// TIA Portal V17 export
// export: Created 2025-06-20T11:32:37.9239786Z, ExportSetting WithDefaults, DisplayName Totally Integrated Automation Portal, DisplayVersion V17 Update 8, DisplayName TIA Portal Openness, DisplayVersion V17 Update 8, DisplayName TIA Portal Version Control Interface, DisplayVersion V17, DisplayName SINAMICS Startdrive Advanced, DisplayVersion V17 SP2, DisplayName SINAMICS Startdrive G110M, G120, G120C, G120D, G120P, G115D, DisplayVersion V17 SP2, DisplayName SINAMICS Startdrive G130, G150, S120, S150, SINAMICS MV, S210, DisplayVersion V17 SP2, DisplayName STEP 7 Professional, DisplayVersion V17 Update 8, DisplayName SINUMERIK ONE STEP 7 Toolbox, DisplayVersion V17 Update 12, DisplayName SINUMERIK ONE PLC Basic Program Plus, DisplayVersion V17 Update 12, DisplayName SINUMERIK 840D sl STEP 7 Toolbox, DisplayVersion V17 Update 12, DisplayName STEP 7 Safety, DisplayVersion V17 Update 6, DisplayName WinCC Advanced, DisplayVersion V17 Update 8
DATA_BLOCK "DB16500_CONNECTION_CALL_MON"   // DB16500
{ S7_Optimized_Access := 'FALSE'; DB_Accessible_From_OPC_UA := 'FALSE' }
VERSION : 0.1
// stored: AutoNumber false, DBAccessibleFromOPCUA false, DBAccessibleFromWebserver false, IsOnlyStoredInLoadMemory false, IsWriteProtectedInAS false
   VAR
      UNIT_1 : Struct
         STA_3_MEAS : Struct
            METHOD : Struct
               NOZZLE_SURFACE_DISTANCE : Struct
                  STATUS : DWord;
                  Connect : DWord;
                  NamespaceGetIndexList : DWord;
                  MethodGetHandleList : DWord;
                  MethodCall : DWord;
                  MethodReleaseHandleList : DWord;
                  Disconnect : DWord;
                  ConnectionGetStatus : DWord;
               END_STRUCT;
               START_LAYER_THICKNESS : Struct
                  STATUS : DWord;
                  Connect : DWord;
                  NamespaceGetIndexList : DWord;
                  MethodGetHandleList : DWord;
                  MethodCall : DWord;
                  MethodReleaseHandleList : DWord;
                  Disconnect : DWord;
                  ConnectionGetStatus : DWord;
               END_STRUCT;
               STOP_LAYER_THICKNESS : Struct
                  STATUS : DWord;
                  Connect : DWord;
                  NamespaceGetIndexList : DWord;
                  MethodGetHandleList : DWord;
                  MethodCall : DWord;
                  MethodReleaseHandleList : DWord;
                  Disconnect : DWord;
                  ConnectionGetStatus : DWord;
               END_STRUCT;
               CALIBRATING : Struct
                  STATUS : DWord;
                  Connect : DWord;
                  NamespaceGetIndexList : DWord;
                  MethodGetHandleList : DWord;
                  MethodCall : DWord;
                  MethodReleaseHandleList : DWord;
                  Disconnect : DWord;
                  ConnectionGetStatus : DWord;
               END_STRUCT;
               RESET : Struct
                  STATUS : DWord;
                  Connect : DWord;
                  NamespaceGetIndexList : DWord;
                  MethodGetHandleList : DWord;
                  MethodCall : DWord;
                  MethodReleaseHandleList : DWord;
                  Disconnect : DWord;
                  ConnectionGetStatus : DWord;
               END_STRUCT;
               READ_VARIABLES : Struct
                  STATUS : DWord;
                  Connect : DWord;
                  NamespaceGetIndexList : DWord;
                  MethodGetHandleList : DWord;
                  MethodCall : DWord;
                  MethodReleaseHandleList : DWord;
                  Disconnect : DWord;
                  ConnectionGetStatus : DWord;
               END_STRUCT;
            END_STRUCT;
            PULSES : Struct
               NOZZLE_SURFACE_DISTANCE : Bool;
               START_LAYER_THICKNESS : Bool;
               STOP_LAYER_THICKNESS : Bool;
               CALIBRATING : Bool;
               RESET : Bool;
               READ_VARIABLES : Bool;
            END_STRUCT;
            TIMERS : Struct
               NOZZLE_SURFACE_DISTANCE : TON_TIME;
               START_LAYER_THICKNESS : TON_TIME;
               STOP_LAYER_THICKNESS : TON_TIME;
               CALIBRATING : TON_TIME;
               RESET : TON_TIME;
               READ_VARIABLES : TON_TIME;
            END_STRUCT;
         END_STRUCT;
         STA_3_COAXIAL : Struct
            METHOD : Struct
               LASER_CALIBRATION : Struct
                  STATUS : DWord;
                  Connect : DWord;
                  NamespaceGetIndexList : DWord;
                  MethodGetHandleList : DWord;
                  MethodCall : DWord;
                  MethodReleaseHandleList : DWord;
                  Disconnect : DWord;
                  ConnectionGetStatus : DWord;
               END_STRUCT;
               NOZZLE_CALIBRATION : Struct
                  STATUS : DWord;
                  Connect : DWord;
                  NamespaceGetIndexList : DWord;
                  MethodGetHandleList : DWord;
                  MethodCall : DWord;
                  MethodReleaseHandleList : DWord;
                  Disconnect : DWord;
                  ConnectionGetStatus : DWord;
               END_STRUCT;
               JET_CALIBRATION : Struct
                  STATUS : DWord;
                  Connect : DWord;
                  NamespaceGetIndexList : DWord;
                  MethodGetHandleList : DWord;
                  MethodCall : DWord;
                  MethodReleaseHandleList : DWord;
                  Disconnect : DWord;
                  ConnectionGetStatus : DWord;
               END_STRUCT;
               CLADDING_CALIBRATION : Struct
                  STATUS : DWord;
                  Connect : DWord;
                  NamespaceGetIndexList : DWord;
                  MethodGetHandleList : DWord;
                  MethodCall : DWord;
                  MethodReleaseHandleList : DWord;
                  Disconnect : DWord;
                  ConnectionGetStatus : DWord;
               END_STRUCT;
               NOZZLE_ANALISIS : Struct
                  STATUS : DWord;
                  Connect : DWord;
                  NamespaceGetIndexList : DWord;
                  MethodGetHandleList : DWord;
                  MethodCall : DWord;
                  MethodReleaseHandleList : DWord;
                  Disconnect : DWord;
                  ConnectionGetStatus : DWord;
               END_STRUCT;
               JET_ANALISIS : Struct
                  STATUS : DWord;
                  Connect : DWord;
                  NamespaceGetIndexList : DWord;
                  MethodGetHandleList : DWord;
                  MethodCall : DWord;
                  MethodReleaseHandleList : DWord;
                  Disconnect : DWord;
                  ConnectionGetStatus : DWord;
               END_STRUCT;
               CLADDING_ANALISIS : Struct
                  STATUS : DWord;
                  Connect : DWord;
                  NamespaceGetIndexList : DWord;
                  MethodGetHandleList : DWord;
                  MethodCall : DWord;
                  MethodReleaseHandleList : DWord;
                  Disconnect : DWord;
                  ConnectionGetStatus : DWord;
               END_STRUCT;
               STOP_METHODS : Struct
                  STATUS : DWord;
                  Connect : DWord;
                  NamespaceGetIndexList : DWord;
                  MethodGetHandleList : DWord;
                  MethodCall : DWord;
                  MethodReleaseHandleList : DWord;
                  Disconnect : DWord;
                  ConnectionGetStatus : DWord;
               END_STRUCT;
               RESET : Struct
                  STATUS : DWord;
                  Connect : DWord;
                  NamespaceGetIndexList : DWord;
                  MethodGetHandleList : DWord;
                  MethodCall : DWord;
                  MethodReleaseHandleList : DWord;
                  Disconnect : DWord;
                  ConnectionGetStatus : DWord;
               END_STRUCT;
               READ_VARIABLES : Struct
                  STATUS : DWord;
                  Connect : DWord;
                  NamespaceGetIndexList : DWord;
                  MethodGetHandleList : DWord;
                  MethodCall : DWord;
                  MethodReleaseHandleList : DWord;
                  Disconnect : DWord;
                  ConnectionGetStatus : DWord;
               END_STRUCT;
            END_STRUCT;
            PULSES : Struct
               LASER_CALIBRATION : Bool;
               NOZZLE_CALIBRATION : Bool;
               JET_CALIBRATION : Bool;
               CLADDING_CALIBRATION : Bool;
               NOZZLE_ANALISIS : Bool;
               JET_ANALISIS : Bool;
               CLADDING_ANALISIS : Bool;
               STOP_METHODS : Bool;
               RESET : Bool;
               READ_VARIABLES : Bool;
            END_STRUCT;
            TIMERS : Struct
               LASER_CALIBRATION : TON_TIME;
               NOZZLE_CALIBRATION : TON_TIME;
               JET_CALIBRATION : TON_TIME;
               CLADDING_CALIBRATION : TON_TIME;
               NOZZLE_ANALISIS : TON_TIME;
               JET_ANALISIS : TON_TIME;
               CLADDING_ANALISIS : TON_TIME;
               STOP_METHODS : TON_TIME;
               RESET : TON_TIME;
               READ_VARIABLES : TON_TIME;
            END_STRUCT;
         END_STRUCT;
      END_STRUCT;
      UNIT_2 : Struct
         STA_2_MEAS : Struct
            METHOD : Struct
               MEASURING : Struct
                  STATUS : DWord;
                  Connect : DWord;
                  NamespaceGetIndexList : DWord;
                  MethodGetHandleList : DWord;
                  MethodCall : DWord;
                  MethodReleaseHandleList : DWord;
                  Disconnect : DWord;
                  ConnectionGetStatus : DWord;
               END_STRUCT;
               CALIBRATING : Struct
                  STATUS : DWord;
                  Connect : DWord;
                  NamespaceGetIndexList : DWord;
                  MethodGetHandleList : DWord;
                  MethodCall : DWord;
                  MethodReleaseHandleList : DWord;
                  Disconnect : DWord;
                  ConnectionGetStatus : DWord;
               END_STRUCT;
               RESET : Struct
                  STATUS : DWord;
                  Connect : DWord;
                  NamespaceGetIndexList : DWord;
                  MethodGetHandleList : DWord;
                  MethodCall : DWord;
                  MethodReleaseHandleList : DWord;
                  Disconnect : DWord;
                  ConnectionGetStatus : DWord;
               END_STRUCT;
               READ_VARIABLES : Struct
                  STATUS : DWord;
                  Connect : DWord;
                  NamespaceGetIndexList : DWord;
                  MethodGetHandleList : DWord;
                  MethodCall : DWord;
                  MethodReleaseHandleList : DWord;
                  Disconnect : DWord;
                  ConnectionGetStatus : DWord;
               END_STRUCT;
            END_STRUCT;
            PULSES : Struct
               MEASURING : Bool;
               CALIBRATING : Bool;
               RESET : Bool;
               READ_VARIABLES : Bool;
            END_STRUCT;
            TIMERS : Struct
               MEASURING : TON_TIME;
               CALIBRATING : TON_TIME;
               RESET : TON_TIME;
               READ_VARIABLES : TON_TIME;
            END_STRUCT;
         END_STRUCT;
         STA_3_COAXIAL : Struct
            METHOD : Struct
               LASER_CALIBRATION : Struct
                  STATUS : DWord;
                  Connect : DWord;
                  NamespaceGetIndexList : DWord;
                  MethodGetHandleList : DWord;
                  MethodCall : DWord;
                  MethodReleaseHandleList : DWord;
                  Disconnect : DWord;
                  ConnectionGetStatus : DWord;
               END_STRUCT;
               NOZZLE_CALIBRATION : Struct
                  STATUS : DWord;
                  Connect : DWord;
                  NamespaceGetIndexList : DWord;
                  MethodGetHandleList : DWord;
                  MethodCall : DWord;
                  MethodReleaseHandleList : DWord;
                  Disconnect : DWord;
                  ConnectionGetStatus : DWord;
               END_STRUCT;
               JET_CALIBRATION : Struct
                  STATUS : DWord;
                  Connect : DWord;
                  NamespaceGetIndexList : DWord;
                  MethodGetHandleList : DWord;
                  MethodCall : DWord;
                  MethodReleaseHandleList : DWord;
                  Disconnect : DWord;
                  ConnectionGetStatus : DWord;
               END_STRUCT;
               CLADDING_CALIBRATION : Struct
                  STATUS : DWord;
                  Connect : DWord;
                  NamespaceGetIndexList : DWord;
                  MethodGetHandleList : DWord;
                  MethodCall : DWord;
                  MethodReleaseHandleList : DWord;
                  Disconnect : DWord;
                  ConnectionGetStatus : DWord;
               END_STRUCT;
               NOZZLE_ANALISIS : Struct
                  STATUS : DWord;
                  Connect : DWord;
                  NamespaceGetIndexList : DWord;
                  MethodGetHandleList : DWord;
                  MethodCall : DWord;
                  MethodReleaseHandleList : DWord;
                  Disconnect : DWord;
                  ConnectionGetStatus : DWord;
               END_STRUCT;
               JET_ANALISIS : Struct
                  STATUS : DWord;
                  Connect : DWord;
                  NamespaceGetIndexList : DWord;
                  MethodGetHandleList : DWord;
                  MethodCall : DWord;
                  MethodReleaseHandleList : DWord;
                  Disconnect : DWord;
                  ConnectionGetStatus : DWord;
               END_STRUCT;
               CLADDING_ANALISIS : Struct
                  STATUS : DWord;
                  Connect : DWord;
                  NamespaceGetIndexList : DWord;
                  MethodGetHandleList : DWord;
                  MethodCall : DWord;
                  MethodReleaseHandleList : DWord;
                  Disconnect : DWord;
                  ConnectionGetStatus : DWord;
               END_STRUCT;
               STOP_METHODS : Struct
                  STATUS : DWord;
                  Connect : DWord;
                  NamespaceGetIndexList : DWord;
                  MethodGetHandleList : DWord;
                  MethodCall : DWord;
                  MethodReleaseHandleList : DWord;
                  Disconnect : DWord;
                  ConnectionGetStatus : DWord;
               END_STRUCT;
               RESET : Struct
                  STATUS : DWord;
                  Connect : DWord;
                  NamespaceGetIndexList : DWord;
                  MethodGetHandleList : DWord;
                  MethodCall : DWord;
                  MethodReleaseHandleList : DWord;
                  Disconnect : DWord;
                  ConnectionGetStatus : DWord;
               END_STRUCT;
               READ_VARIABLES : Struct
                  STATUS : DWord;
                  Connect : DWord;
                  NamespaceGetIndexList : DWord;
                  MethodGetHandleList : DWord;
                  MethodCall : DWord;
                  MethodReleaseHandleList : DWord;
                  Disconnect : DWord;
                  ConnectionGetStatus : DWord;
               END_STRUCT;
            END_STRUCT;
            PULSES : Struct
               LASER_CALIBRATION : Bool;
               NOZZLE_CALIBRATION : Bool;
               JET_CALIBRATION : Bool;
               CLADDING_CALIBRATION : Bool;
               NOZZLE_ANALISIS : Bool;
               JET_ANALISIS : Bool;
               CLADDING_ANALISIS : Bool;
               STOP_METHODS : Bool;
               RESET : Bool;
               READ_VARIABLES : Bool;
            END_STRUCT;
            TIMERS : Struct
               LASER_CALIBRATION : TON_TIME;
               NOZZLE_CALIBRATION : TON_TIME;
               JET_CALIBRATION : TON_TIME;
               CLADDING_CALIBRATION : TON_TIME;
               NOZZLE_ANALISIS : TON_TIME;
               JET_ANALISIS : TON_TIME;
               CLADDING_ANALISIS : TON_TIME;
               STOP_METHODS : TON_TIME;
               RESET : TON_TIME;
               READ_VARIABLES : TON_TIME;
            END_STRUCT;
         END_STRUCT;
         STA_3_MEAS : Struct
            METHOD : Struct
               NOZZLE_SURFACE_DISTANCE : Struct
                  STATUS : DWord;
                  Connect : DWord;
                  NamespaceGetIndexList : DWord;
                  MethodGetHandleList : DWord;
                  MethodCall : DWord;
                  MethodReleaseHandleList : DWord;
                  Disconnect : DWord;
                  ConnectionGetStatus : DWord;
               END_STRUCT;
               START_LAYER_THICKNESS : Struct
                  STATUS : DWord;
                  Connect : DWord;
                  NamespaceGetIndexList : DWord;
                  MethodGetHandleList : DWord;
                  MethodCall : DWord;
                  MethodReleaseHandleList : DWord;
                  Disconnect : DWord;
                  ConnectionGetStatus : DWord;
               END_STRUCT;
               STOP_LAYER_THICKNESS : Struct
                  STATUS : DWord;
                  Connect : DWord;
                  NamespaceGetIndexList : DWord;
                  MethodGetHandleList : DWord;
                  MethodCall : DWord;
                  MethodReleaseHandleList : DWord;
                  Disconnect : DWord;
                  ConnectionGetStatus : DWord;
               END_STRUCT;
               CALIBRATING : Struct
                  STATUS : DWord;
                  Connect : DWord;
                  NamespaceGetIndexList : DWord;
                  MethodGetHandleList : DWord;
                  MethodCall : DWord;
                  MethodReleaseHandleList : DWord;
                  Disconnect : DWord;
                  ConnectionGetStatus : DWord;
               END_STRUCT;
               RESET : Struct
                  STATUS : DWord;
                  Connect : DWord;
                  NamespaceGetIndexList : DWord;
                  MethodGetHandleList : DWord;
                  MethodCall : DWord;
                  MethodReleaseHandleList : DWord;
                  Disconnect : DWord;
                  ConnectionGetStatus : DWord;
               END_STRUCT;
               READ_VARIABLES : Struct
                  STATUS : DWord;
                  Connect : DWord;
                  NamespaceGetIndexList : DWord;
                  MethodGetHandleList : DWord;
                  MethodCall : DWord;
                  MethodReleaseHandleList : DWord;
                  Disconnect : DWord;
                  ConnectionGetStatus : DWord;
               END_STRUCT;
            END_STRUCT;
            PULSES : Struct
               NOZZLE_SURFACE_DISTANCE : Bool;
               START_LAYER_THICKNESS : Bool;
               STOP_LAYER_THICKNESS : Bool;
               CALIBRATING : Bool;
               RESET : Bool;
               READ_VARIABLES : Bool;
            END_STRUCT;
            TIMERS : Struct
               NOZZLE_SURFACE_DISTANCE : TON_TIME;
               START_LAYER_THICKNESS : TON_TIME;
               STOP_LAYER_THICKNESS : TON_TIME;
               CALIBRATING : TON_TIME;
               RESET : TON_TIME;
               READ_VARIABLES : TON_TIME;
            END_STRUCT;
         END_STRUCT;
      END_STRUCT;
      UNIT_3 : Struct
         FACE_R : Struct
            METHOD : Struct
               MEASURING : Struct
                  STATUS : DWord;
                  Connect : DWord;
                  NamespaceGetIndexList : DWord;
                  MethodGetHandleList : DWord;
                  MethodCall : DWord;
                  MethodReleaseHandleList : DWord;
                  Disconnect : DWord;
                  ConnectionGetStatus : DWord;
               END_STRUCT;
               CALIBRATING : Struct
                  STATUS : DWord;
                  Connect : DWord;
                  NamespaceGetIndexList : DWord;
                  MethodGetHandleList : DWord;
                  MethodCall : DWord;
                  MethodReleaseHandleList : DWord;
                  Disconnect : DWord;
                  ConnectionGetStatus : DWord;
               END_STRUCT;
               RESET : Struct
                  STATUS : DWord;
                  Connect : DWord;
                  NamespaceGetIndexList : DWord;
                  MethodGetHandleList : DWord;
                  MethodCall : DWord;
                  MethodReleaseHandleList : DWord;
                  Disconnect : DWord;
                  ConnectionGetStatus : DWord;
               END_STRUCT;
               READ_VARIABLES : Struct
                  STATUS : DWord;
                  Connect : DWord;
                  NamespaceGetIndexList : DWord;
                  MethodGetHandleList : DWord;
                  MethodCall : DWord;
                  MethodReleaseHandleList : DWord;
                  Disconnect : DWord;
                  ConnectionGetStatus : DWord;
               END_STRUCT;
            END_STRUCT;
            PULSES : Struct
               MEASURING : Bool;
               CALIBRATING : Bool;
               RESET : Bool;
               READ_VARIABLES : Bool;
            END_STRUCT;
            TIMERS : Struct
               MEASURING : TON_TIME;
               CALIBRATING : TON_TIME;
               RESET : TON_TIME;
               READ_VARIABLES : TON_TIME;
            END_STRUCT;
         END_STRUCT;
         FACE_N : Struct
            METHOD : Struct
               MEASURING : Struct
                  STATUS : DWord;
                  Connect : DWord;
                  NamespaceGetIndexList : DWord;
                  MethodGetHandleList : DWord;
                  MethodCall : DWord;
                  MethodReleaseHandleList : DWord;
                  Disconnect : DWord;
                  ConnectionGetStatus : DWord;
               END_STRUCT;
               CALIBRATING : Struct
                  STATUS : DWord;
                  Connect : DWord;
                  NamespaceGetIndexList : DWord;
                  MethodGetHandleList : DWord;
                  MethodCall : DWord;
                  MethodReleaseHandleList : DWord;
                  Disconnect : DWord;
                  ConnectionGetStatus : DWord;
               END_STRUCT;
               RESET : Struct
                  STATUS : DWord;
                  Connect : DWord;
                  NamespaceGetIndexList : DWord;
                  MethodGetHandleList : DWord;
                  MethodCall : DWord;
                  MethodReleaseHandleList : DWord;
                  Disconnect : DWord;
                  ConnectionGetStatus : DWord;
               END_STRUCT;
               READ_VARIABLES : Struct
                  STATUS : DWord;
                  Connect : DWord;
                  NamespaceGetIndexList : DWord;
                  MethodGetHandleList : DWord;
                  MethodCall : DWord;
                  MethodReleaseHandleList : DWord;
                  Disconnect : DWord;
                  ConnectionGetStatus : DWord;
               END_STRUCT;
            END_STRUCT;
            PULSES : Struct
               MEASURING : Bool;
               CALIBRATING : Bool;
               RESET : Bool;
               READ_VARIABLES : Bool;
            END_STRUCT;
            TIMERS : Struct
               MEASURING : TON_TIME;
               CALIBRATING : TON_TIME;
               RESET : TON_TIME;
               READ_VARIABLES : TON_TIME;
            END_STRUCT;
         END_STRUCT;
      END_STRUCT;
   END_VAR
BEGIN
   UNIT_1.STA_3_MEAS.TIMERS.NOZZLE_SURFACE_DISTANCE.PT := T#10s;
   UNIT_1.STA_3_MEAS.TIMERS.START_LAYER_THICKNESS.PT := T#10s;
   UNIT_1.STA_3_MEAS.TIMERS.STOP_LAYER_THICKNESS.PT := T#10s;
   UNIT_1.STA_3_MEAS.TIMERS.CALIBRATING.PT := T#10s;
   UNIT_1.STA_3_MEAS.TIMERS.RESET.PT := T#10s;
   UNIT_1.STA_3_MEAS.TIMERS.READ_VARIABLES.PT := T#10s;
   UNIT_1.STA_3_COAXIAL.TIMERS.LASER_CALIBRATION.PT := T#10s;
   UNIT_1.STA_3_COAXIAL.TIMERS.NOZZLE_CALIBRATION.PT := T#10s;
   UNIT_1.STA_3_COAXIAL.TIMERS.JET_CALIBRATION.PT := T#10s;
   UNIT_1.STA_3_COAXIAL.TIMERS.CLADDING_CALIBRATION.PT := T#10s;
   UNIT_1.STA_3_COAXIAL.TIMERS.NOZZLE_ANALISIS.PT := T#10s;
   UNIT_1.STA_3_COAXIAL.TIMERS.JET_ANALISIS.PT := T#10s;
   UNIT_1.STA_3_COAXIAL.TIMERS.CLADDING_ANALISIS.PT := T#10s;
   UNIT_1.STA_3_COAXIAL.TIMERS.STOP_METHODS.PT := T#10s;
   UNIT_1.STA_3_COAXIAL.TIMERS.RESET.PT := T#10s;
   UNIT_1.STA_3_COAXIAL.TIMERS.READ_VARIABLES.PT := T#10s;
   UNIT_2.STA_3_MEAS.TIMERS.NOZZLE_SURFACE_DISTANCE.PT := T#10s;
   UNIT_2.STA_3_MEAS.TIMERS.START_LAYER_THICKNESS.PT := T#10s;
   UNIT_2.STA_3_MEAS.TIMERS.STOP_LAYER_THICKNESS.PT := T#10s;
   UNIT_2.STA_3_MEAS.TIMERS.CALIBRATING.PT := T#10s;
   UNIT_2.STA_3_MEAS.TIMERS.RESET.PT := T#10s;
   UNIT_2.STA_3_MEAS.TIMERS.READ_VARIABLES.PT := T#10s;
END_DATA_BLOCK
